{attribute 'pack_mode' := '1'}
TYPE
  ST_OpcUa_LrealPointWrite :
  STRUCT
    ErrorCode : UDINT;
    Value : LREAL;
  END_STRUCT
END_TYPE

(* stored: Version 1.1.0.1, ProductVersion 3.1.4024.9
   DUT ST_OpcUa_LrealPointWrite: Id {cfe1670a-f5b1-4b0f-8f1d-63c2503aef6e} *)
